Omron Sysmac Studio project Palletizing_Application_2 (Sysmac Studio 1.40.0.64008, StandardProject)

# Controller new_Controller_0: NJ501-1400 version 1.18
Units and slaves: Power Supply : NJ-Px3001; CPU : NJ501-1400
Task PrimaryTask (priority 4, period or condition 2000): TM_Modbus, TM_Movements_Connection, TM_Modbus_Connection, TM_Movements
Library TM_Commands 1.2.1 (contents left out)
Library TM_Modbus 1.1.0 (contents left out)

VAR_GLOBAL
    StartProgram : BOOL;
    CableConnected : BOOL;
    ListenNode_Connect_Connected : BOOL;
    ListenNode_Connect_TCP_Socket : _sSOCKET;
    MTCP_Connect_Connected : BOOL;
    MTCP_Connect_TCP_Socket : _sSOCKET;
END_VAR

PROGRAM TM_Modbus
VAR
    Enable : BOOL;
    DU_Enable : R_TRIG;
    NStep : INT;
    TON_Instance : TON;
    TM_Status_Instance : TM_Status;
    TM_Stop_Instance : TM_Stop;
    TM_ErrorCode_Instance : TM_ErrorCode;
    TM_PlayPause_Instance : TM_PlayPause;
    TM_ErrorCode_Execute : BOOL;
    TM_ErrorCode_Done : BOOL;
    TM_ErrorCode_Busy : BOOL;
    TM_ErrorCode_Error : BOOL;
    TM_ErrorCode_ErrorID : WORD;
    TM_Status_Execute : BOOL;
    TM_Status_Done : BOOL;
    TM_PlayPause_Execute : BOOL;
    TM_PlayPause_Done : BOOL;
    TM_PlayPause_Busy : BOOL;
    TM_PlayPause_Error : BOOL;
    TM_PlayPause_ErrorID : WORD;
    TM_Stop_Execute : BOOL;
    TM_Stop_Done : BOOL;
    TM_Stop_Busy : BOOL;
    TM_Stop_Error : BOOL;
    TM_Stop_ErrorID : WORD;
    TM_Status_Busy : BOOL;
    TM_Status_Error : BOOL;
    TM_Status_ErrorID : WORD;
    TM_ReadPosition_Instance : TM_ReadPosition;
    TM_ReadPosition_Execute : BOOL;
    TM_ReadPosition_Done : BOOL;
    TM_ReadPosition_Busy : BOOL;
    TM_ReadPosition_Error : BOOL;
    TM_ReadPosition_ErrorID : WORD;
    TM_ErrorCode_TMErrorCode : DINT;
    TM_Status_TMEditing : BOOL;
    TM_Status_TMError : BOOL;
    TM_Status_TMPaused : BOOL;
    TM_Status_TMRunning : BOOL;
    TM_PlayPauseButton : BOOL;
    TM_StopButton : BOOL;
    TM_ReadPosition_X : REAL;
    TM_ReadPosition_Y : REAL;
    TM_ReadPosition_Z : REAL;
    TM_ReadPosition_RX : REAL;
    TM_ReadPosition_RY : REAL;
    TM_ReadPosition_RZ : REAL;
END_VAR
VAR_EXTERNAL
    StartProgram : BOOL;
    CableConnected : BOOL;
    MTCP_Connect_TCP_Socket : _sSOCKET;
    MTCP_Connect_Connected : BOOL;
END_VAR
DU_Enable(Clk:=Enable);

Enable:=StartProgram;

IF DU_Enable.Q THEN
	
	NStep:=0;
	
END_IF;

IF Enable AND MTCP_Connect_Connected THEN
	
	CASE NStep OF
		
		0:
			IF TM_PlayPauseButton THEN
				NStep:=100;
			ELSIF TM_StopButton THEN
				NStep:=200;
			ELSE
				NStep:=300;
			END_IF;
		100:
			TM_PlayPause_Execute:=FALSE;
			TON_Instance.PT:=T#3s;
			TON_Instance.In:=FALSE;
			IF NOT TM_PlayPause_Done AND NOT TM_PlayPause_Error AND NOT TON_Instance.Q THEN
				NStep:=110;
			END_IF;
		110:
			TM_PlayPause_Execute:=TRUE;
			TON_Instance.In:=TRUE;
			IF TM_PlayPause_Done THEN
				CableConnected:=TRUE;
				TM_PlayPauseButton:=FALSE;
				NStep:=300;
			ELSIF (TM_PlayPause_Error AND (TM_PlayPause_ErrorID=16#2003 OR TM_PlayPause_ErrorID=16#2006)) THEN
				NStep:=300;
				CableConnected:=FALSE;
			ELSIF TON_Instance.Q THEN
				NStep:=100;
			END_IF;
		200:
			TM_Stop_Execute:=FALSE;
			TON_Instance.PT:=T#3s;
			TON_Instance.In:=FALSE;
			IF NOT TM_Stop_Done AND NOT TM_Stop_Error AND NOT TON_Instance.Q THEN
				NStep:=210;
			END_IF;
		210:
			TM_Stop_Execute:=TRUE;
			TON_Instance.In:=TRUE;
			IF TM_Stop_Done THEN
				TM_StopButton:=FALSE;
				CableConnected:=TRUE;
				NStep:=300;
			ELSIF (TM_Stop_Error AND (TM_Stop_ErrorID=16#2003 OR TM_Stop_ErrorID=16#2006)) THEN
				NStep:=300;
				CableConnected:=FALSE;
			ELSIF TON_Instance.Q THEN
				NStep:=200;
			END_IF;
		300:
			TM_Status_Execute:=FALSE;
			TON_Instance.PT:=T#3s;
			TON_Instance.In:=FALSE;
			IF NOT TM_Status_Done AND NOT TM_Status_Error AND NOT TON_Instance.Q THEN
				NStep:=310;
			END_IF;
		310:
			TM_Status_Execute:=TRUE;
			TON_Instance.In:=TRUE;
			IF TM_Status_Done THEN
				NStep:=400;
				CableConnected:=TRUE;
			ELSIF TM_Status_Error AND (TM_Status_ErrorID=16#2003 OR  TM_Status_ErrorID=16#2006) THEN
				NStep:=300;
				CableConnected:=FALSE;
			ELSIF TON_Instance.Q THEN
				NStep:=300;
			END_IF;
		400:
			TM_ErrorCode_Execute:=FALSE;
			TON_Instance.PT:=T#3s;
			TON_Instance.In:=FALSE;
			IF NOT TM_ErrorCode_Done AND NOT TM_ErrorCode_Error AND NOT TON_Instance.Q THEN
				NStep:=410;
			END_IF;
		410:
			TM_ErrorCode_Execute:=TRUE;
			TON_Instance.In:=TRUE;
			IF TM_ErrorCode_Done THEN
				CableConnected:=TRUE;
				NStep:=500;
			ELSIF (TM_ErrorCode_Error AND (TM_ErrorCode_ErrorID=16#2003 OR TM_ErrorCode_ErrorID=16#2006)) THEN
				NStep:=400;
				CableConnected:=FALSE;
			ELSIF TON_Instance.Q THEN
				NStep:=400;
			END_IF;
		500:
			TM_ReadPosition_Execute:=FALSE;
			TON_Instance.PT:=T#3s;
			TON_Instance.In:=FALSE;
			IF NOT TM_ReadPosition_Done AND NOT TM_ReadPosition_Error AND NOT TON_Instance.Q THEN
				NStep:=510;
			END_IF;
		510:
			TM_ReadPosition_Execute:=TRUE;
			TON_Instance.In:=TRUE;
			IF TM_ReadPosition_Done THEN
				CableConnected:=TRUE;
				NStep:=600;
			ELSIF (TM_ReadPosition_Error AND (TM_ReadPosition_ErrorID=16#2003 OR TM_ReadPosition_ErrorID=16#2006)) THEN
				NStep:=500;
				CableConnected:=FALSE;
			ELSIF TON_Instance.Q THEN
				NStep:=500;
			END_IF;
		600:
			TON_Instance.In:=FALSE;
			TON_Instance.PT:=T#1s;
			IF (NOT TON_Instance.Q) THEN
				NStep:=610;
			END_IF;
		610:
			TON_Instance.In:=TRUE;
			IF TON_Instance.Q THEN
				NStep:=0;
			END_IF;		
		
	END_CASE;
	
END_IF;

TON_Instance();

TM_ErrorCode_Instance(
	Execute:=TM_ErrorCode_Execute,
	Socket:=MTCP_Connect_TCP_Socket,
	Done=>TM_ErrorCode_Done,
	TMErrorCode=>TM_ErrorCode_TMErrorCode,
	Busy=>TM_ErrorCode_Busy,
	Error=>TM_ErrorCode_Error,
	ErrorID=>TM_ErrorCode_ErrorID
);

TM_Status_Instance(
	Execute:=TM_Status_Execute,
	Socket:=MTCP_Connect_TCP_Socket,
	Done=>TM_Status_Done,
	TMRunning=>TM_Status_TMRunning,
	TMEditing=>TM_Status_TMEditing,
	TMError=>TM_Status_TMError,
	TMPaused=>TM_Status_TMPaused,
	Busy=>TM_Status_Busy,
	Error=>TM_Status_Error,
	ErrorID=>TM_Status_ErrorID
);

TM_PlayPause_Instance(
	Execute:=TM_PlayPause_Execute,
	Socket:=MTCP_Connect_TCP_Socket,
	Done=>TM_PlayPause_Done,
	Busy=>TM_PlayPause_Busy,
	Error=>TM_PlayPause_Error,
	ErrorID=>TM_PlayPause_ErrorID
);

TM_Stop_Instance(
	Execute:=TM_Stop_Execute,
	Socket:=MTCP_Connect_TCP_Socket,
	Done=>TM_Stop_Done,
	Busy=>TM_Stop_Busy,
	Error=>TM_Stop_Error,
	ErrorID=>TM_Stop_ErrorID
);

TM_ReadPosition_Instance(
	Execute:=TM_ReadPosition_Execute,
	Socket:=MTCP_Connect_TCP_Socket,
	Done=>TM_ReadPosition_Done,
	Busy=>TM_ReadPosition_Busy,
	Error=>TM_ReadPosition_Error,
	ErrorID=>TM_ReadPosition_ErrorID,
	X=>TM_ReadPosition_X,
	Y=>TM_ReadPosition_Y,
	Z=>TM_ReadPosition_Z,
	RX=>TM_ReadPosition_RX,
	RY=>TM_ReadPosition_RY,
	RZ=>TM_ReadPosition_RZ
);
END_PROGRAM

PROGRAM TM_Movements_Connection
VAR
    ListenNode_Connect_Instance : ListenNode_Connect;
    ListenNode_Connect_Enable : BOOL;
    ListenNode_Connect_IPaddress : STRING[16];
    ListenNode_Connect_Port : UINT;
    ListenNode_Connect_Connect : BOOL;
    ListenNode_Connect_Error : BOOL;
    ListenNode_Connect_ErrorID : WORD;
    ListenNode_Connect_EtnConnError : BOOL;
    ListenNode_Connect_Socket_Status : _eCONNECTION_STATE;
END_VAR
VAR_EXTERNAL
    ListenNode_Connect_Connected : BOOL;
    ListenNode_Connect_TCP_Socket : _sSOCKET;
    StartProgram : BOOL;
END_VAR
ListenNode_Connect_Enable:=TRUE;
ListenNode_Connect_IPaddress:='192.168.250.30';
ListenNode_Connect_Port:=5890;

ListenNode_Connect_Connect:=StartProgram;

ListenNode_Connect_Instance(
	Enable:=ListenNode_Connect_Enable,
	IPaddress:=ListenNode_Connect_IPaddress,
	Port:=ListenNode_Connect_Port,
	Connect:=ListenNode_Connect_Connect,
	Connected=>ListenNode_Connect_Connected,
	Error=>ListenNode_Connect_Error,
	ErrorID=>ListenNode_Connect_ErrorID,
	EtnConnError=>ListenNode_Connect_EtnConnError,
	TCP_Socket=>ListenNode_Connect_TCP_Socket,
	Socket_Status=>ListenNode_Connect_Socket_Status
);
END_PROGRAM

PROGRAM TM_Modbus_Connection
VAR
    MTCP_Connect_Instance : MTCP_Connect;
    MTCP_Connect_Enable : BOOL;
    MTCP_Connect_Port : UINT;
    MTCP_Connect_Connect : BOOL;
    MTCP_Connect_Error : BOOL;
    MTCP_Connect_ErrorID : WORD;
    MTCP_Connect_EtnConnError : BOOL;
    MTCP_Connect_Socket_Status : _eCONNECTION_STATE;
    MTCP_Connect_IPaddress : STRING[16];
END_VAR
VAR_EXTERNAL
    StartProgram : BOOL;
    MTCP_Connect_Connected : BOOL;
    MTCP_Connect_TCP_Socket : _sSOCKET;
END_VAR
MTCP_Connect_Enable:=TRUE;
MTCP_Connect_IPaddress:='192.168.250.30';
MTCP_Connect_Port:=502;

MTCP_Connect_Connect:=StartProgram;

MTCP_Connect_Instance(
	Enable:=MTCP_Connect_Enable,
	IPaddress:=MTCP_Connect_IPaddress,
	Port:=MTCP_Connect_Port,
	Connect:=MTCP_Connect_Connect,
	Connected=>MTCP_Connect_Connected,
	Error=>MTCP_Connect_Error,
	ErrorID=>MTCP_Connect_ErrorID,
	EtnConnError=>MTCP_Connect_EtnConnError,
	TCP_Socket=>MTCP_Connect_TCP_Socket,
	Socket_Status=>MTCP_Connect_Socket_Status
);
END_PROGRAM

PROGRAM TM_Movements
VAR
    TM_ChangeLoad_Instance : TM_ChangeLoad;
    TM_ChangeTCP_Instance : TM_ChangeTCP;
    TM_MovCmd_Instance : TM_MovCmd;
    TM_MovCmd_Done : BOOL;
    TM_MovCmd_Busy : BOOL;
    TM_MovCmd_Error : BOOL;
    TM_MovCmd_ErrorID : WORD;
    TM_MovCmd_Execute : BOOL;
    TM_MovCmd_Movement : STRING[256];
    TM_MovCmd_DataFormat : STRING[256];
    DD_ListenNode_Connect_Connected : F_TRIG;
    TM_MovCmd_Point : STRING[256];
    TM_MovCmd_Speed : INT;
    TM_MovCmd_AccelTime : INT;
    TM_MovCmd_Blending : INT;
    TM_MovCmd_PrecisePos : BOOL;
    TM_MovCmd_RobotPose : STRING[256];
    TM_MovCmd_Command : STRING[256];
    TM_MovCmd_ActivateExit : BOOL;
    TM_MovCmd_CommandID : INT;
    Enable : BOOL;
    DU_Enable : R_TRIG;
    TM_ChangeBase_Busy : BOOL;
    TM_ChangeBase_Done : BOOL;
    TM_ChangeBase_Error : BOOL;
    TM_ChangeBase_ErrorID : WORD;
    TM_ChangeBase_Execute : BOOL;
    TM_ChangeBase_Base : STRING[256];
    TM_ChangeBase_ActivateExit : BOOL;
    TM_ChangeBase_CommandID : INT;
    TM_ChangeLoad_Execute : BOOL;
    TM_ChangeLoad_Busy : BOOL;
    TM_ChangeLoad_Done : BOOL;
    TM_ChangeLoad_Error : BOOL;
    TM_ChangeLoad_ErrorID : WORD;
    TM_ChangeLoad_Payload : STRING[256];
    TM_ChangeLoad_ActivateExit : BOOL;
    TM_ChangeLoad_CommandID : INT;
    TM_ChangeTCP_Busy : BOOL;
    TM_ChangeTCP_Done : BOOL;
    TM_ChangeTCP_Error : BOOL;
    TM_ChangeTCP_ErrorID : WORD;
    TM_ChangeTCP_Execute : BOOL;
    TM_ChangeTCP_TCP : STRING[256];
    TM_ChangeTCP_Weight : STRING[256];
    TM_ChangeTCP_MomInertia : STRING[256];
    TM_ChangeTCP_RefFrame : STRING[256];
    TM_ChangeTCP_ActivateExit : BOOL;
    TM_ChangeTCP_CommandID : INT;
    TM_CircleCmd_Done : BOOL;
    TM_CircleCmd_Busy : BOOL;
    TM_CircleCmd_Error : BOOL;
    TM_CircleCmd_ErrorID : WORD;
    TM_CircleCmd_Execute : BOOL;
    TM_CircleCmd_DataFormat : STRING[256];
    TM_CircleCmd_ArcPoint : STRING[256];
    TM_CircleCmd_EndArcPoint : STRING[256];
    TM_CircleCmd_Speed : INT;
    TM_CircleCmd_AccelTime : INT;
    TM_CircleCmd_Blending : INT;
    TM_CircleCmd_ArcAngle : INT;
    TM_CircleCmd_PrecisePos : BOOL;
    TM_CircleCmd_Command : STRING[256];
    TM_CircleCmd_ActivateExit : BOOL;
    TM_CircleCmd_CommandID : INT;
    PickPoint : STRING[256];
    PalletFirstPoint : STRING[256];
    StartPoint : STRING[256];
    PalletSecondPoint : STRING[256];
    PalletThirdPoint : STRING[256];
    PalletFourthPoint : STRING[256];
    MovementIndicatorStage : INT;
    DownRelative : STRING[256];
    HighRelative : STRING[256];
    TM_ChangeBase_Command : STRING[256];
    TM_ChangeLoad_Command : STRING[256];
    TM_ChangeTCP_Command : STRING[256];
    DD_CableConnected : F_TRIG;
    TM_MovCmd_ListenNode : STRING[256];
    Stage : INT;
    TM_MovCmd_TimeOutET : TIME;
    TM_MovCmd_Enable : BOOL;
    TM_ChangeTCP_Enable : BOOL;
    TM_ChangeTCP_ListenNode : STRING[256];
    TM_ChangeTCP_TimeOutET : TIME;
    TM_ChangeLoad_Enable : BOOL;
    TM_ChangeLoad_ListenNode : STRING[256];
    TM_ChangeLoad_TimeOutET : TIME;
    TM_CircleCmd_Instance : TM_CircleCmd;
    TM_ChangeBase_Instance : TM_ChangeBase;
    TM_ChangeBase_Enable : BOOL;
    TM_CircleCmd_Enable : BOOL;
    TM_CircleCmd_ListenNode : STRING[256];
    TM_CircleCmd_TimeOutET : TIME;
    TM_ChangeBase_ListenNode : STRING[256];
    TM_ChangeBase_TimeOutET : TIME;
END_VAR
VAR_EXTERNAL
    StartProgram : BOOL;
    CableConnected : BOOL;
    ListenNode_Connect_Connected : BOOL;
    ListenNode_Connect_TCP_Socket : _sSOCKET;
END_VAR
DU_Enable(Clk:=Enable);
DD_ListenNode_Connect_Connected(Clk:=ListenNode_Connect_Connected);
DD_CableConnected(Clk:=CableConnected);

Enable:=StartProgram;

IF DU_Enable.Q THEN
	
	Stage:=0;
	MovementIndicatorStage:=0;
	
	PickPoint:='400,100,400,180,0,90';
	PalletFirstPoint:='200,-200,400,180,0,90';
	PalletSecondPoint:='200,-400,400,180,0,90';
	PalletThirdPoint:='400,-200,400,180,0,90';
	PalletFourthPoint:='400,-400,400,180,0,90';
	StartPoint:='400,0,500,150,0,90';
	DownRelative:='0,0,-100,0,0,0';
	HighRelative:='0,0,100,0,0,0';
	
END_IF;

IF DD_ListenNode_Connect_Connected.Q OR DD_CableConnected.Q THEN //connection closed or cable disconnected.
	
	Stage:=MovementIndicatorStage;
	
END_IF;

IF Enable AND ListenNode_Connect_Connected AND CableConnected THEN	//the PLC program is enabled and there is connection with listen node and the cable is connected
	
	CASE Stage OF
		
		//-----------------------------------------------------------TCP Selection--------------------------------------------------
		0:
			TM_ChangeTCP_Enable:=FALSE;
			IF (NOT TM_ChangeTCP_Done) AND (NOT TM_ChangeTCP_Error) AND (NOT TM_ChangeTCP_Busy) THEN
				Stage:=1; 
			END_IF;
		1:
			TM_ChangeTCP_Enable:=TRUE;	
			TM_ChangeTCP_ActivateExit:=TRUE;
			TM_ChangeTCP_CommandID:=1;
			TM_ChangeTCP_Execute:=FALSE;
			TM_ChangeTCP_ListenNode:='Listen1';
			TM_ChangeTCP_TCP:='DefinedTool';
			TM_ChangeTCP_Command:='var_i=10';
			TM_ChangeTCP_Weight:='';
			TM_ChangeTCP_MomInertia:='';
			TM_ChangeTCP_RefFrame:='';
			TM_ChangeLoad_Payload:='';
			IF (NOT TM_ChangeTCP_Done) AND (NOT TM_ChangeTCP_Error) THEN
				Stage:=2;
			END_IF;
		2:
			TM_ChangeTCP_Execute:=TRUE;
			IF TM_ChangeTCP_Done THEN
				Stage:=10;
			ELSIF TM_ChangeTCP_Error THEN
				Stage:=9999;
			END_IF;
		//-----------------------------------------------------------Program Stages--------------------------------------------------------------
		10:
			TM_MovCmd_Enable:=FALSE;
			MovementIndicatorStage:=Stage;
			IF (NOT TM_MovCmd_Done) AND (NOT TM_MovCmd_Error) AND (NOT TM_MovCmd_Busy) THEN
				Stage:=11;
			END_IF;
		11:
			TM_MovCmd_Enable:=TRUE;
			TM_MovCmd_Movement:='PTP';
			TM_MovCmd_DataFormat:='CPP';
			TM_MovCmd_Point:=StartPoint;
			TM_MovCmd_Speed:=30;
			TM_MovCmd_AccelTime:=200;
			TM_MovCmd_Blending:=100;
			TM_MovCmd_PrecisePos:=1;
			TM_MovCmd_RobotPose:='';
			TM_MovCmd_Command:='var_i=40';
			TM_MovCmd_ActivateExit:=TRUE;
			TM_MovCmd_CommandID:=1;
			TM_MovCmd_Execute:=FALSE;
			TM_MovCmd_ListenNode:='Listen1';
			IF (NOT TM_MovCmd_Done) AND (NOT TM_MovCmd_Error) THEN
				Stage:=12;
			END_IF;
		12:
			TM_MovCmd_Execute:=TRUE;
			IF TM_MovCmd_Done THEN
				Stage:=20;
			ELSIF TM_MovCmd_Error THEN
				Stage:=9999;
			END_IF;
		20:
			TM_MovCmd_Enable:=FALSE;
			MovementIndicatorStage:=Stage;
			IF (NOT TM_MovCmd_Done) AND (NOT TM_MovCmd_Error) AND (NOT TM_MovCmd_Busy) THEN
				Stage:=21;
			END_IF;
		21:			
			TM_MovCmd_Enable:=TRUE;
			TM_MovCmd_Movement:='Line';
			TM_MovCmd_DataFormat:='CPR';
			TM_MovCmd_Point:=StartPoint;
			TM_MovCmd_Speed:=30;
			TM_MovCmd_AccelTime:=200;
			TM_MovCmd_Blending:=100;
			TM_MovCmd_PrecisePos:=1;
			TM_MovCmd_RobotPose:='';
			TM_MovCmd_Command:='var_i=30';
			TM_MovCmd_ActivateExit:=TRUE;
			TM_MovCmd_CommandID:=1;
			TM_MovCmd_Execute:=FALSE;
			TM_MovCmd_ListenNode:='Listen1';
			IF (NOT TM_MovCmd_Done) AND (NOT TM_MovCmd_Error) THEN
				Stage:=22;
			END_IF;	
		22:
			TM_MovCmd_Execute:=TRUE;
			IF TM_MovCmd_Done THEN
				Stage:=30;
			ELSIF TM_MovCmd_Error THEN
				Stage:=9999;
			END_IF;
		30:
			TM_MovCmd_Enable:=FALSE;
			MovementIndicatorStage:=Stage;
			IF (NOT TM_MovCmd_Done) AND (NOT TM_MovCmd_Error) AND (NOT TM_MovCmd_Busy) THEN
				Stage:=31;
			END_IF;
		31:			
			TM_MovCmd_Enable:=TRUE;
			TM_MovCmd_Movement:='Line';
			TM_MovCmd_DataFormat:='CPR';
			TM_MovCmd_Point:=PickPoint;
			TM_MovCmd_Speed:=30;
			TM_MovCmd_AccelTime:=200;
			TM_MovCmd_Blending:=100;
			TM_MovCmd_PrecisePos:=1;
			TM_MovCmd_RobotPose:='';
			TM_MovCmd_Command:='var_i=10';
			TM_MovCmd_ActivateExit:=FALSE;
			TM_MovCmd_CommandID:=1;
			TM_MovCmd_Execute:=FALSE;
			TM_MovCmd_ListenNode:='Listen1';
			IF (NOT TM_MovCmd_Done) AND (NOT TM_MovCmd_Error) THEN
				Stage:=32;
			END_IF;			
		32:
			TM_MovCmd_Execute:=TRUE;
			IF TM_MovCmd_Done THEN
				Stage:=40;
			ELSIF TM_MovCmd_Error THEN
				Stage:=9999;
			END_IF;
		40:
			TM_MovCmd_Enable:=FALSE;
			IF (NOT TM_MovCmd_Done) AND (NOT TM_MovCmd_Error) AND (NOT TM_MovCmd_Busy) THEN
				Stage:=41;
			END_IF;
		41:			
			TM_MovCmd_Enable:=TRUE;
			TM_MovCmd_Movement:='Move_Line';
			TM_MovCmd_DataFormat:='CPP';
			TM_MovCmd_Point:=DownRelative;
			TM_MovCmd_Speed:=30;
			TM_MovCmd_AccelTime:=200;
			TM_MovCmd_Blending:=100;
			TM_MovCmd_PrecisePos:=1;
			TM_MovCmd_RobotPose:='';
			TM_MovCmd_Command:='var_i=10';
			TM_MovCmd_ActivateExit:=TRUE;
			TM_MovCmd_CommandID:=2;
			TM_MovCmd_Execute:=FALSE;
			TM_MovCmd_ListenNode:='Listen1';
			IF (NOT TM_MovCmd_Done) AND (NOT TM_MovCmd_Error) THEN
				Stage:=42;
			END_IF;
		42:
			TM_MovCmd_Execute:=TRUE;
			IF TM_MovCmd_Done THEN
				Stage:=50;
			ELSIF TM_MovCmd_Error THEN
				Stage:=9999;
			END_IF;
		50:
			TM_ChangeLoad_Enable:=FALSE;
			IF (NOT TM_ChangeLoad_Done) AND (NOT TM_ChangeLoad_Error) AND (NOT TM_ChangeLoad_Busy) THEN
				Stage:=51;
			END_IF;
		51:
			TM_ChangeLoad_Enable:=TRUE;	 
			TM_ChangeLoad_ActivateExit:=TRUE;
			TM_ChangeLoad_CommandID:=1;
			TM_ChangeLoad_Execute:=FALSE;
			TM_ChangeLoad_ListenNode:='Listen1';
			TM_ChangeLoad_Command:='var_i=20';
			TM_ChangeLoad_Payload:='0.2';
			IF (NOT TM_ChangeLoad_Done) AND (NOT TM_ChangeLoad_Error) THEN
				Stage:=52;
			END_IF;
		52:
			TM_ChangeLoad_Execute:=TRUE;
			IF TM_ChangeLoad_Done THEN
				Stage:=60;
			ELSIF TM_ChangeLoad_Error THEN
				Stage:=9999;
			END_IF;			
		60:
			TM_MovCmd_Enable:=FALSE;
			IF (NOT TM_MovCmd_Done) AND (NOT TM_MovCmd_Error) AND (NOT TM_MovCmd_Busy) THEN
				Stage:=61;
			END_IF;	
		61:
			TM_MovCmd_Enable:=TRUE;
			TM_MovCmd_Movement:='Move_Line';
			TM_MovCmd_DataFormat:='CPP';
			TM_MovCmd_Point:=HighRelative;
			TM_MovCmd_Speed:=30;
			TM_MovCmd_AccelTime:=200;
			TM_MovCmd_Blending:=100;
			TM_MovCmd_PrecisePos:=1;
			TM_MovCmd_RobotPose:='';
			TM_MovCmd_Command:='var_i=10';
			TM_MovCmd_ActivateExit:=TRUE;
			TM_MovCmd_CommandID:=2;
			TM_MovCmd_Execute:=FALSE;
			TM_MovCmd_ListenNode:='Listen1';
			IF (NOT TM_MovCmd_Done) AND (NOT TM_MovCmd_Error) THEN
				Stage:=62;
			END_IF;
		62:
			TM_MovCmd_Execute:=TRUE;
			IF TM_MovCmd_Done THEN
				Stage:=70;
			ELSIF TM_MovCmd_Error THEN
				Stage:=9999;
			END_IF;
		70:
			TM_MovCmd_Enable:=FALSE;
			MovementIndicatorStage:=Stage;
			IF (NOT TM_MovCmd_Done) AND (NOT TM_MovCmd_Error) AND (NOT TM_MovCmd_Busy) THEN
				Stage:=71;
			END_IF;	
		71:
			TM_MovCmd_Enable:=TRUE;
			TM_MovCmd_Movement:='Line';
			TM_MovCmd_DataFormat:='CPR';
			TM_MovCmd_Point:=PalletFirstPoint;
			TM_MovCmd_Speed:=30;
			TM_MovCmd_AccelTime:=200;
			TM_MovCmd_Blending:=100;
			TM_MovCmd_PrecisePos:=1;
			TM_MovCmd_RobotPose:='';
			TM_MovCmd_Command:='var_i=10';
			TM_MovCmd_ActivateExit:=FALSE;
			TM_MovCmd_CommandID:=1;
			TM_MovCmd_Execute:=FALSE;
			TM_MovCmd_ListenNode:='Listen1';
			IF (NOT TM_MovCmd_Done) AND (NOT TM_MovCmd_Error) THEN
				Stage:=72;
			END_IF;
		72:
			TM_MovCmd_Execute:=TRUE;
			IF TM_MovCmd_Done THEN
				Stage:=80;
			ELSIF TM_MovCmd_Error THEN
				Stage:=9999;
			END_IF;
		80:
			TM_MovCmd_Enable:=FALSE;
			IF (NOT TM_MovCmd_Done) AND (NOT TM_MovCmd_Error) AND (NOT TM_MovCmd_Busy) THEN
				Stage:=81;
			END_IF;	
		81:
			TM_MovCmd_Enable:=TRUE;
			TM_MovCmd_Movement:='Move_Line';
			TM_MovCmd_DataFormat:='CPP';
			TM_MovCmd_Point:=DownRelative;
			TM_MovCmd_Speed:=30;
			TM_MovCmd_AccelTime:=200;
			TM_MovCmd_Blending:=100;
			TM_MovCmd_PrecisePos:=1;
			TM_MovCmd_RobotPose:='';
			TM_MovCmd_Command:='var_i=10';
			TM_MovCmd_ActivateExit:=TRUE;
			TM_MovCmd_CommandID:=2;
			TM_MovCmd_Execute:=FALSE;
			TM_MovCmd_ListenNode:='Listen1';
			IF (NOT TM_MovCmd_Done) AND (NOT TM_MovCmd_Error) THEN
				Stage:=82;
			END_IF;
		82:
			TM_MovCmd_Execute:=TRUE;
			IF TM_MovCmd_Done THEN
				Stage:=90;
			ELSIF TM_MovCmd_Error THEN
				Stage:=9999;
			END_IF;
		90:
			TM_ChangeLoad_Enable:=FALSE;
			IF (NOT TM_ChangeLoad_Done) AND (NOT TM_ChangeLoad_Error) AND (NOT TM_ChangeLoad_Busy) THEN
				Stage:=91;
			END_IF;
		91:
			TM_ChangeLoad_Enable:=TRUE;	 
			TM_ChangeLoad_ActivateExit:=TRUE;
			TM_ChangeLoad_CommandID:=1;
			TM_ChangeLoad_Execute:=FALSE;
			TM_ChangeLoad_ListenNode:='Listen1';
			TM_ChangeLoad_Command:='var_i=30';
			TM_ChangeLoad_Payload:='0';
			IF (NOT TM_ChangeLoad_Done) AND (NOT TM_ChangeLoad_Error) THEN
				Stage:=92;
			END_IF;
		92:
			TM_ChangeLoad_Execute:=TRUE;
			IF TM_ChangeLoad_Done THEN
				Stage:=100;
			ELSIF TM_ChangeLoad_Error THEN
				Stage:=9999;
			END_IF;
		100:
			TM_MovCmd_Enable:=FALSE;
			IF (NOT TM_MovCmd_Done) AND (NOT TM_MovCmd_Error) AND (NOT TM_MovCmd_Busy) THEN
				Stage:=101;
			END_IF;	
		101:
			TM_MovCmd_Enable:=TRUE;
			TM_MovCmd_Movement:='Move_Line';
			TM_MovCmd_DataFormat:='CPP';
			TM_MovCmd_Point:=HighRelative;
			TM_MovCmd_Speed:=30;
			TM_MovCmd_AccelTime:=200;
			TM_MovCmd_Blending:=100;
			TM_MovCmd_PrecisePos:=1;
			TM_MovCmd_RobotPose:='';
			TM_MovCmd_Command:='var_i=10';
			TM_MovCmd_ActivateExit:=TRUE;
			TM_MovCmd_CommandID:=2;
			TM_MovCmd_Execute:=FALSE;
			TM_MovCmd_ListenNode:='Listen1';
			IF (NOT TM_MovCmd_Done) AND (NOT TM_MovCmd_Error) THEN
				Stage:=102;
			END_IF;
		102:
			TM_MovCmd_Execute:=TRUE;
			IF TM_MovCmd_Done THEN
				Stage:=110;
			ELSIF TM_MovCmd_Error THEN
				Stage:=9999;
			END_IF;
		110:
			TM_MovCmd_Enable:=FALSE;
			MovementIndicatorStage:=Stage;
			IF (NOT TM_MovCmd_Done) AND (NOT TM_MovCmd_Error) AND (NOT TM_MovCmd_Busy) THEN
				Stage:=111;
			END_IF;	
		111:
			TM_MovCmd_Enable:=TRUE;
			TM_MovCmd_Movement:='Line';
			TM_MovCmd_DataFormat:='CPR';
			TM_MovCmd_Point:=PickPoint;
			TM_MovCmd_Speed:=30;
			TM_MovCmd_AccelTime:=200;
			TM_MovCmd_Blending:=100;
			TM_MovCmd_PrecisePos:=1;
			TM_MovCmd_RobotPose:='';
			TM_MovCmd_Command:='var_i=10';
			TM_MovCmd_ActivateExit:=FALSE;
			TM_MovCmd_CommandID:=1;
			TM_MovCmd_Execute:=FALSE;
			TM_MovCmd_ListenNode:='Listen1';
			IF (NOT TM_MovCmd_Done) AND (NOT TM_MovCmd_Error) THEN
				Stage:=112;
			END_IF;
		112:
			TM_MovCmd_Execute:=TRUE;
			IF TM_MovCmd_Done THEN
				Stage:=120;
			ELSIF TM_MovCmd_Error THEN
				Stage:=9999;
			END_IF;
		120:
			TM_MovCmd_Enable:=FALSE;
			IF (NOT TM_MovCmd_Done) AND (NOT TM_MovCmd_Error) AND (NOT TM_MovCmd_Busy) THEN
				Stage:=121;
			END_IF;	
		121:
			TM_MovCmd_Enable:=TRUE;
			TM_MovCmd_Movement:='Move_Line';
			TM_MovCmd_DataFormat:='CPP';
			TM_MovCmd_Point:=DownRelative;
			TM_MovCmd_Speed:=30;
			TM_MovCmd_AccelTime:=200;
			TM_MovCmd_Blending:=100;
			TM_MovCmd_PrecisePos:=1;
			TM_MovCmd_RobotPose:='';
			TM_MovCmd_Command:='var_i=10';
			TM_MovCmd_ActivateExit:=TRUE;
			TM_MovCmd_CommandID:=2;
			TM_MovCmd_Execute:=FALSE;
			TM_MovCmd_ListenNode:='Listen1';
			IF (NOT TM_MovCmd_Done) AND (NOT TM_MovCmd_Error) THEN
				Stage:=122;
			END_IF;
		122:
			TM_MovCmd_Execute:=TRUE;
			IF TM_MovCmd_Done THEN
				Stage:=130;
			ELSIF TM_MovCmd_Error THEN
				Stage:=9999;
			END_IF;
		130:
			TM_ChangeLoad_Enable:=FALSE;
			IF (NOT TM_ChangeLoad_Done) AND (NOT TM_ChangeLoad_Error) AND (NOT TM_ChangeLoad_Busy) THEN
				Stage:=131;
			END_IF;
		131:
			TM_ChangeLoad_Enable:=TRUE;	 
			TM_ChangeLoad_ActivateExit:=TRUE;
			TM_ChangeLoad_CommandID:=1;
			TM_ChangeLoad_Execute:=FALSE;
			TM_ChangeLoad_ListenNode:='Listen1';
			TM_ChangeLoad_Command:='var_i=20';
			TM_ChangeLoad_Payload:='0.2';
			IF (NOT TM_ChangeLoad_Done) AND (NOT TM_ChangeLoad_Error) THEN
				Stage:=132;
			END_IF;
		132:
			TM_ChangeLoad_Execute:=TRUE;
			IF TM_ChangeLoad_Done THEN
				Stage:=140;
			ELSIF TM_ChangeLoad_Error THEN
				Stage:=9999;
			END_IF;
		140:
			TM_MovCmd_Enable:=FALSE;
			IF (NOT TM_MovCmd_Done) AND (NOT TM_MovCmd_Error) AND (NOT TM_MovCmd_Busy) THEN
				Stage:=141;
			END_IF;
		141:
			TM_MovCmd_Enable:=TRUE;
			TM_MovCmd_Movement:='Move_Line';
			TM_MovCmd_DataFormat:='CPP';
			TM_MovCmd_Point:=HighRelative;
			TM_MovCmd_Speed:=30;
			TM_MovCmd_AccelTime:=200;
			TM_MovCmd_Blending:=100;
			TM_MovCmd_PrecisePos:=1;
			TM_MovCmd_RobotPose:='';
			TM_MovCmd_Command:='var_i=10';
			TM_MovCmd_ActivateExit:=TRUE;
			TM_MovCmd_CommandID:=2;
			TM_MovCmd_Execute:=FALSE;
			TM_MovCmd_ListenNode:='Listen1';
			IF (NOT TM_MovCmd_Done) AND (NOT TM_MovCmd_Error) THEN
				Stage:=142;
			END_IF;
		142:
			TM_MovCmd_Execute:=TRUE;
			IF TM_MovCmd_Done THEN
				Stage:=150;
			ELSIF TM_MovCmd_Error THEN
				Stage:=9999;
			END_IF;
		150:
			TM_MovCmd_Enable:=FALSE;
			MovementIndicatorStage:=Stage;
			IF (NOT TM_MovCmd_Done) AND (NOT TM_MovCmd_Error) AND (NOT TM_MovCmd_Busy) THEN
				Stage:=151;
			END_IF;
		151:
			TM_MovCmd_Enable:=TRUE;
			TM_MovCmd_Movement:='Line';
			TM_MovCmd_DataFormat:='CPR';
			TM_MovCmd_Point:=PalletSecondPoint;
			TM_MovCmd_Speed:=30;
			TM_MovCmd_AccelTime:=200;
			TM_MovCmd_Blending:=100;
			TM_MovCmd_PrecisePos:=1;
			TM_MovCmd_RobotPose:='';
			TM_MovCmd_Command:='var_i=10';
			TM_MovCmd_ActivateExit:=FALSE;
			TM_MovCmd_CommandID:=1;
			TM_MovCmd_Execute:=FALSE;
			TM_MovCmd_ListenNode:='Listen1';
			IF (NOT TM_MovCmd_Done) AND (NOT TM_MovCmd_Error) THEN
				Stage:=152;
			END_IF;
		152:
			TM_MovCmd_Execute:=TRUE;
			IF TM_MovCmd_Done THEN
				Stage:=160;
			ELSIF TM_MovCmd_Error THEN
				Stage:=9999;
			END_IF;
		160:
			TM_MovCmd_Enable:=FALSE;
			IF (NOT TM_MovCmd_Done) AND (NOT TM_MovCmd_Error) AND (NOT TM_MovCmd_Busy) THEN
				Stage:=161;
			END_IF;	
		161:
			TM_MovCmd_Enable:=TRUE;
			TM_MovCmd_Movement:='Move_Line';
			TM_MovCmd_DataFormat:='CPP';
			TM_MovCmd_Point:=DownRelative;
			TM_MovCmd_Speed:=30;
			TM_MovCmd_AccelTime:=200;
			TM_MovCmd_Blending:=100;
			TM_MovCmd_PrecisePos:=1;
			TM_MovCmd_RobotPose:='';
			TM_MovCmd_Command:='var_i=10';
			TM_MovCmd_ActivateExit:=TRUE;
			TM_MovCmd_CommandID:=2;
			TM_MovCmd_Execute:=FALSE;
			TM_MovCmd_ListenNode:='Listen1';
			IF (NOT TM_MovCmd_Done) AND (NOT TM_MovCmd_Error) THEN
				Stage:=162;
			END_IF;
		162:
			TM_MovCmd_Execute:=TRUE;
			IF TM_MovCmd_Done THEN
				Stage:=170;
			ELSIF TM_MovCmd_Error THEN
				Stage:=9999;
			END_IF;
		170:
			TM_ChangeLoad_Enable:=FALSE;
			IF (NOT TM_ChangeLoad_Done) AND (NOT TM_ChangeLoad_Error) AND (NOT TM_ChangeLoad_Busy) THEN
				Stage:=171;
			END_IF;
		171:
			TM_ChangeLoad_Enable:=TRUE;	 
			TM_ChangeLoad_ActivateExit:=TRUE;
			TM_ChangeLoad_CommandID:=1;
			TM_ChangeLoad_Execute:=FALSE;
			TM_ChangeLoad_ListenNode:='Listen1';
			TM_ChangeLoad_Command:='var_i=30';
			TM_ChangeLoad_Payload:='0';
			IF (NOT TM_ChangeLoad_Done) AND (NOT TM_ChangeLoad_Error) THEN
				Stage:=172;
			END_IF;
		172:
			TM_ChangeLoad_Execute:=TRUE;
			IF TM_ChangeLoad_Done THEN
				Stage:=180;
			ELSIF TM_ChangeLoad_Error THEN
				Stage:=9999;
			END_IF;
		180:
			TM_MovCmd_Enable:=FALSE;
			IF (NOT TM_MovCmd_Done) AND (NOT TM_MovCmd_Error) AND (NOT TM_MovCmd_Busy) THEN
				Stage:=181;
			END_IF;	
		181:
			TM_MovCmd_Enable:=TRUE;
			TM_MovCmd_Movement:='Move_Line';
			TM_MovCmd_DataFormat:='CPP';
			TM_MovCmd_Point:=HighRelative;
			TM_MovCmd_Speed:=30;
			TM_MovCmd_AccelTime:=200;
			TM_MovCmd_Blending:=100;
			TM_MovCmd_PrecisePos:=1;
			TM_MovCmd_RobotPose:='';
			TM_MovCmd_Command:='var_i=10';
			TM_MovCmd_ActivateExit:=TRUE;
			TM_MovCmd_CommandID:=2;
			TM_MovCmd_Execute:=FALSE;
			TM_MovCmd_ListenNode:='Listen1';
			IF (NOT TM_MovCmd_Done) AND (NOT TM_MovCmd_Error) THEN
				Stage:=182;
			END_IF;
		182:
			TM_MovCmd_Execute:=TRUE;
			IF TM_MovCmd_Done THEN
				Stage:=190;
			ELSIF TM_MovCmd_Error THEN
				Stage:=9999;
			END_IF;
		190:
			TM_MovCmd_Enable:=FALSE;
			MovementIndicatorStage:=Stage;
			IF (NOT TM_MovCmd_Done) AND (NOT TM_MovCmd_Error) AND (NOT TM_MovCmd_Busy) THEN
				Stage:=191;
			END_IF;	
		191:
			TM_MovCmd_Enable:=TRUE;
			TM_MovCmd_Movement:='Line';
			TM_MovCmd_DataFormat:='CPR';
			TM_MovCmd_Point:=PickPoint;
			TM_MovCmd_Speed:=30;
			TM_MovCmd_AccelTime:=200;
			TM_MovCmd_Blending:=100;
			TM_MovCmd_PrecisePos:=1;
			TM_MovCmd_RobotPose:='';
			TM_MovCmd_Command:='var_i=10';
			TM_MovCmd_ActivateExit:=FALSE;
			TM_MovCmd_CommandID:=1;
			TM_MovCmd_Execute:=FALSE;
			TM_MovCmd_ListenNode:='Listen1';
			IF (NOT TM_MovCmd_Done) AND (NOT TM_MovCmd_Error) THEN
				Stage:=192;
			END_IF;
		192:
			TM_MovCmd_Execute:=TRUE;
			IF TM_MovCmd_Done THEN
				Stage:=200;
			ELSIF TM_MovCmd_Error THEN
				Stage:=9999;
			END_IF;
		200:
			TM_MovCmd_Enable:=FALSE;
			IF (NOT TM_MovCmd_Done) AND (NOT TM_MovCmd_Error) AND (NOT TM_MovCmd_Busy) THEN
				Stage:=201;
			END_IF;	
		201:
			TM_MovCmd_Enable:=TRUE;
			TM_MovCmd_Movement:='Move_Line';
			TM_MovCmd_DataFormat:='CPP';
			TM_MovCmd_Point:=DownRelative;
			TM_MovCmd_Speed:=30;
			TM_MovCmd_AccelTime:=200;
			TM_MovCmd_Blending:=100;
			TM_MovCmd_PrecisePos:=1;
			TM_MovCmd_RobotPose:='';
			TM_MovCmd_Command:='var_i=10';
			TM_MovCmd_ActivateExit:=TRUE;
			TM_MovCmd_CommandID:=2;
			TM_MovCmd_Execute:=FALSE;
			TM_MovCmd_ListenNode:='Listen1';
			IF (NOT TM_MovCmd_Done) AND (NOT TM_MovCmd_Error) THEN
				Stage:=202;
			END_IF;
		202:
			TM_MovCmd_Execute:=TRUE;
			IF TM_MovCmd_Done THEN
				Stage:=210;
			ELSIF TM_MovCmd_Error THEN
				Stage:=9999;
			END_IF;
		210:
			TM_ChangeLoad_Enable:=FALSE;
			IF (NOT TM_ChangeLoad_Done) AND (NOT TM_ChangeLoad_Error) AND (NOT TM_ChangeLoad_Busy) THEN
				Stage:=211;
			END_IF;
		211:
			TM_ChangeLoad_Enable:=TRUE;	 
			TM_ChangeLoad_ActivateExit:=TRUE;
			TM_ChangeLoad_CommandID:=1;
			TM_ChangeLoad_Execute:=FALSE;
			TM_ChangeLoad_ListenNode:='Listen1';
			TM_ChangeLoad_Command:='var_i=20';
			TM_ChangeLoad_Payload:='0.2';
			IF (NOT TM_ChangeLoad_Done) AND (NOT TM_ChangeLoad_Error) THEN
				Stage:=212;
			END_IF;
		212:
			TM_ChangeLoad_Execute:=TRUE;
			IF TM_ChangeLoad_Done THEN
				Stage:=220;
			ELSIF TM_ChangeLoad_Error THEN
				Stage:=9999;
			END_IF;
		220:
			TM_MovCmd_Enable:=FALSE;
			IF (NOT TM_MovCmd_Done) AND (NOT TM_MovCmd_Error) AND (NOT TM_MovCmd_Busy) THEN
				Stage:=221;
			END_IF;
		221:
			TM_MovCmd_Enable:=TRUE;
			TM_MovCmd_Movement:='Move_Line';
			TM_MovCmd_DataFormat:='CPP';
			TM_MovCmd_Point:=HighRelative;
			TM_MovCmd_Speed:=30;
			TM_MovCmd_AccelTime:=200;
			TM_MovCmd_Blending:=100;
			TM_MovCmd_PrecisePos:=1;
			TM_MovCmd_RobotPose:='';
			TM_MovCmd_Command:='var_i=10';
			TM_MovCmd_ActivateExit:=TRUE;
			TM_MovCmd_CommandID:=2;
			TM_MovCmd_Execute:=FALSE;
			TM_MovCmd_ListenNode:='Listen1';
			IF (NOT TM_MovCmd_Done) AND (NOT TM_MovCmd_Error) THEN
				Stage:=222;
			END_IF;
		222:
			TM_MovCmd_Execute:=TRUE;
			IF TM_MovCmd_Done THEN
				Stage:=230;
			ELSIF TM_MovCmd_Error THEN
				Stage:=9999;
			END_IF;
		230:
			TM_MovCmd_Enable:=FALSE;
			MovementIndicatorStage:=Stage;
			IF (NOT TM_MovCmd_Done) AND (NOT TM_MovCmd_Error) AND (NOT TM_MovCmd_Busy) THEN
				Stage:=231;
			END_IF;
		231:
			TM_MovCmd_Enable:=TRUE;
			TM_MovCmd_Movement:='Line';
			TM_MovCmd_DataFormat:='CPR';
			TM_MovCmd_Point:=PalletThirdPoint;
			TM_MovCmd_Speed:=30;
			TM_MovCmd_AccelTime:=200;
			TM_MovCmd_Blending:=100;
			TM_MovCmd_PrecisePos:=1;
			TM_MovCmd_RobotPose:='';
			TM_MovCmd_Command:='var_i=10';
			TM_MovCmd_ActivateExit:=FALSE;
			TM_MovCmd_CommandID:=1;
			TM_MovCmd_Execute:=FALSE;
			TM_MovCmd_ListenNode:='Listen1';
			IF (NOT TM_MovCmd_Done) AND (NOT TM_MovCmd_Error) THEN
				Stage:=232;
			END_IF;
		232:
			TM_MovCmd_Execute:=TRUE;
			IF TM_MovCmd_Done THEN
				Stage:=240;
			ELSIF TM_MovCmd_Error THEN
				Stage:=9999;
			END_IF;
		240:
			TM_MovCmd_Enable:=FALSE;
			IF (NOT TM_MovCmd_Done) AND (NOT TM_MovCmd_Error) AND (NOT TM_MovCmd_Busy) THEN
				Stage:=241;
			END_IF;
		241:
			TM_MovCmd_Enable:=TRUE;
			TM_MovCmd_Movement:='Move_Line';
			TM_MovCmd_DataFormat:='CPP';
			TM_MovCmd_Point:=DownRelative;
			TM_MovCmd_Speed:=30;
			TM_MovCmd_AccelTime:=200;
			TM_MovCmd_Blending:=100;
			TM_MovCmd_PrecisePos:=1;
			TM_MovCmd_RobotPose:='';
			TM_MovCmd_Command:='var_i=10';
			TM_MovCmd_ActivateExit:=TRUE;
			TM_MovCmd_CommandID:=2;
			TM_MovCmd_Execute:=FALSE;
			TM_MovCmd_ListenNode:='Listen1';
			IF (NOT TM_MovCmd_Done) AND (NOT TM_MovCmd_Error) THEN
				Stage:=242;
			END_IF;
		242:
			TM_MovCmd_Execute:=TRUE;
			IF TM_MovCmd_Done THEN
				Stage:=250;
			ELSIF TM_MovCmd_Error THEN
				Stage:=9999;
			END_IF;
		250:
			TM_ChangeLoad_Enable:=FALSE;
			IF (NOT TM_ChangeLoad_Done) AND (NOT TM_ChangeLoad_Error) AND (NOT TM_ChangeLoad_Busy) THEN
				Stage:=251;
			END_IF;
		251:
			TM_ChangeLoad_Enable:=TRUE;	 
			TM_ChangeLoad_ActivateExit:=TRUE;
			TM_ChangeLoad_CommandID:=1;
			TM_ChangeLoad_Execute:=FALSE;
			TM_ChangeLoad_ListenNode:='Listen1';
			TM_ChangeLoad_Command:='var_i=30';
			TM_ChangeLoad_Payload:='0';
			IF (NOT TM_ChangeLoad_Done) AND (NOT TM_ChangeLoad_Error) THEN
				Stage:=252;
			END_IF;
		252:
			TM_ChangeLoad_Execute:=TRUE;
			IF TM_ChangeLoad_Done THEN
				Stage:=260;
			ELSIF TM_ChangeLoad_Error THEN
				Stage:=9999;
			END_IF;
		260:
			TM_MovCmd_Enable:=FALSE;
			IF (NOT TM_MovCmd_Done) AND (NOT TM_MovCmd_Error) AND (NOT TM_MovCmd_Busy) THEN
				Stage:=261;
			END_IF;
		261:
			TM_MovCmd_Enable:=TRUE;
			TM_MovCmd_Movement:='Move_Line';
			TM_MovCmd_DataFormat:='CPP';
			TM_MovCmd_Point:=HighRelative;
			TM_MovCmd_Speed:=30;
			TM_MovCmd_AccelTime:=200;
			TM_MovCmd_Blending:=100;
			TM_MovCmd_PrecisePos:=1;
			TM_MovCmd_RobotPose:='';
			TM_MovCmd_Command:='var_i=10';
			TM_MovCmd_ActivateExit:=TRUE;
			TM_MovCmd_CommandID:=2;
			TM_MovCmd_Execute:=FALSE;
			TM_MovCmd_ListenNode:='Listen1';
			IF (NOT TM_MovCmd_Done) AND (NOT TM_MovCmd_Error) THEN
				Stage:=262;
			END_IF;
		262:
			TM_MovCmd_Execute:=TRUE;
			IF TM_MovCmd_Done THEN
				Stage:=270;
			ELSIF TM_MovCmd_Error THEN
				Stage:=9999;
			END_IF;
		270:
			TM_MovCmd_Enable:=FALSE;
			MovementIndicatorStage:=Stage;
			IF (NOT TM_MovCmd_Done) AND (NOT TM_MovCmd_Error) AND (NOT TM_MovCmd_Busy) THEN
				Stage:=271;
			END_IF;
		271:
			TM_MovCmd_Enable:=TRUE;
			TM_MovCmd_Movement:='Line';
			TM_MovCmd_DataFormat:='CPR';
			TM_MovCmd_Point:=PickPoint;
			TM_MovCmd_Speed:=30;
			TM_MovCmd_AccelTime:=200;
			TM_MovCmd_Blending:=100;
			TM_MovCmd_PrecisePos:=1;
			TM_MovCmd_RobotPose:='';
			TM_MovCmd_Command:='var_i=10';
			TM_MovCmd_ActivateExit:=FALSE;
			TM_MovCmd_CommandID:=1;
			TM_MovCmd_Execute:=FALSE;
			TM_MovCmd_ListenNode:='Listen1';
			IF (NOT TM_MovCmd_Done) AND (NOT TM_MovCmd_Error) THEN
				Stage:=272;
			END_IF;
		272:
			TM_MovCmd_Execute:=TRUE;
			IF TM_MovCmd_Done THEN
				Stage:=280;
			ELSIF TM_MovCmd_Error THEN
				Stage:=9999;
			END_IF;
		280:
			TM_MovCmd_Enable:=FALSE;
			IF (NOT TM_MovCmd_Done) AND (NOT TM_MovCmd_Error) AND (NOT TM_MovCmd_Busy) THEN
				Stage:=281;
			END_IF;
		281:
			TM_MovCmd_Enable:=TRUE;
			TM_MovCmd_Movement:='Move_Line';
			TM_MovCmd_DataFormat:='CPP';
			TM_MovCmd_Point:=DownRelative;
			TM_MovCmd_Speed:=30;
			TM_MovCmd_AccelTime:=200;
			TM_MovCmd_Blending:=100;
			TM_MovCmd_PrecisePos:=1;
			TM_MovCmd_RobotPose:='';
			TM_MovCmd_Command:='var_i=10';
			TM_MovCmd_ActivateExit:=TRUE;
			TM_MovCmd_CommandID:=2;
			TM_MovCmd_Execute:=FALSE;
			TM_MovCmd_ListenNode:='Listen1';
			IF (NOT TM_MovCmd_Done) AND (NOT TM_MovCmd_Error) THEN
				Stage:=282;
			END_IF;
		282:
			TM_MovCmd_Execute:=TRUE;
			IF TM_MovCmd_Done THEN
				Stage:=290;
			ELSIF TM_MovCmd_Error THEN
				Stage:=9999;
			END_IF;
		290:
			TM_ChangeLoad_Enable:=FALSE;
			IF (NOT TM_ChangeLoad_Done) AND (NOT TM_ChangeLoad_Error) AND (NOT TM_ChangeLoad_Busy) THEN
				Stage:=291;
			END_IF;
		291:
			TM_ChangeLoad_Enable:=TRUE;	 
			TM_ChangeLoad_ActivateExit:=TRUE;
			TM_ChangeLoad_CommandID:=1;
			TM_ChangeLoad_Execute:=FALSE;
			TM_ChangeLoad_ListenNode:='Listen1';
			TM_ChangeLoad_Command:='var_i=20';
			TM_ChangeLoad_Payload:='0.2';
			IF (NOT TM_ChangeLoad_Done) AND (NOT TM_ChangeLoad_Error) THEN
				Stage:=292;
			END_IF;
		292:
			TM_ChangeLoad_Execute:=TRUE;
			IF TM_ChangeLoad_Done THEN
				Stage:=300;
			ELSIF TM_ChangeLoad_Error THEN
				Stage:=9999;
			END_IF;
		300:
			TM_MovCmd_Enable:=FALSE;
			IF (NOT TM_MovCmd_Done) AND (NOT TM_MovCmd_Error) AND (NOT TM_MovCmd_Busy) THEN
				Stage:=301;
			END_IF;
		301:
			TM_MovCmd_Enable:=TRUE;
			TM_MovCmd_Movement:='Move_Line';
			TM_MovCmd_DataFormat:='CPP';
			TM_MovCmd_Point:=HighRelative;
			TM_MovCmd_Speed:=30;
			TM_MovCmd_AccelTime:=200;
			TM_MovCmd_Blending:=100;
			TM_MovCmd_PrecisePos:=1;
			TM_MovCmd_RobotPose:='';
			TM_MovCmd_Command:='var_i=10';
			TM_MovCmd_ActivateExit:=TRUE;
			TM_MovCmd_CommandID:=2;
			TM_MovCmd_Execute:=FALSE;
			TM_MovCmd_ListenNode:='Listen1';
			IF (NOT TM_MovCmd_Done) AND (NOT TM_MovCmd_Error) THEN
				Stage:=302;
			END_IF;
		302:
			TM_MovCmd_Execute:=TRUE;
			IF TM_MovCmd_Done THEN
				Stage:=310;
			ELSIF TM_MovCmd_Error THEN
				Stage:=9999;
			END_IF;
		310:
			TM_MovCmd_Enable:=FALSE;
			MovementIndicatorStage:=Stage;
			IF (NOT TM_MovCmd_Done) AND (NOT TM_MovCmd_Error) AND (NOT TM_MovCmd_Busy) THEN
				Stage:=311;
			END_IF;
		311:
			TM_MovCmd_Enable:=TRUE;
			TM_MovCmd_Movement:='Line';
			TM_MovCmd_DataFormat:='CPR';
			TM_MovCmd_Point:=PalletFourthPoint;
			TM_MovCmd_Speed:=30;
			TM_MovCmd_AccelTime:=200;
			TM_MovCmd_Blending:=100;
			TM_MovCmd_PrecisePos:=1;
			TM_MovCmd_RobotPose:='';
			TM_MovCmd_Command:='var_i=10';
			TM_MovCmd_ActivateExit:=FALSE;
			TM_MovCmd_CommandID:=1;
			TM_MovCmd_Execute:=FALSE;
			TM_MovCmd_ListenNode:='Listen1';
			IF (NOT TM_MovCmd_Done) AND (NOT TM_MovCmd_Error) THEN
				Stage:=312;
			END_IF;
		312:
			TM_MovCmd_Execute:=TRUE;
			IF TM_MovCmd_Done THEN
				Stage:=320;
			ELSIF TM_MovCmd_Error THEN
				Stage:=9999;
			END_IF;
		320:
			TM_MovCmd_Enable:=FALSE;
			IF (NOT TM_MovCmd_Done) AND (NOT TM_MovCmd_Error) AND (NOT TM_MovCmd_Busy) THEN
				Stage:=321;
			END_IF;
		321:
			TM_MovCmd_Enable:=TRUE;
			TM_MovCmd_Movement:='Move_Line';
			TM_MovCmd_DataFormat:='CPP';
			TM_MovCmd_Point:=DownRelative;
			TM_MovCmd_Speed:=30;
			TM_MovCmd_AccelTime:=200;
			TM_MovCmd_Blending:=100;
			TM_MovCmd_PrecisePos:=1;
			TM_MovCmd_RobotPose:='';
			TM_MovCmd_Command:='var_i=10';
			TM_MovCmd_ActivateExit:=TRUE;
			TM_MovCmd_CommandID:=2;
			TM_MovCmd_Execute:=FALSE;
			TM_MovCmd_ListenNode:='Listen1';
			IF (NOT TM_MovCmd_Done) AND (NOT TM_MovCmd_Error) THEN
				Stage:=322;
			END_IF;
		322:
			TM_MovCmd_Execute:=TRUE;
			IF TM_MovCmd_Done THEN
				Stage:=330;
			ELSIF TM_MovCmd_Error THEN
				Stage:=9999;
			END_IF;
		330:
			TM_ChangeLoad_Enable:=FALSE;
			IF (NOT TM_ChangeLoad_Done) AND (NOT TM_ChangeLoad_Error) AND (NOT TM_ChangeLoad_Busy) THEN
				Stage:=331;
			END_IF;
		331:
			TM_ChangeLoad_Enable:=TRUE;	 
			TM_ChangeLoad_ActivateExit:=TRUE;
			TM_ChangeLoad_CommandID:=1;
			TM_ChangeLoad_Execute:=FALSE;
			TM_ChangeLoad_ListenNode:='Listen1';
			TM_ChangeLoad_Command:='var_i=30';
			TM_ChangeLoad_Payload:='0';
			IF (NOT TM_ChangeLoad_Done) AND (NOT TM_ChangeLoad_Error) THEN
				Stage:=332;
			END_IF;
		332:
			TM_ChangeLoad_Execute:=TRUE;
			IF TM_ChangeLoad_Done THEN
				Stage:=340;
			ELSIF TM_ChangeLoad_Error THEN
				Stage:=9999;
			END_IF;
		340:
			TM_MovCmd_Enable:=FALSE;
			IF (NOT TM_MovCmd_Done) AND (NOT TM_MovCmd_Error) AND (NOT TM_MovCmd_Busy) THEN
				Stage:=341;
			END_IF;
		341:
			TM_MovCmd_Enable:=TRUE;
			TM_MovCmd_Movement:='Move_Line';
			TM_MovCmd_DataFormat:='CPP';
			TM_MovCmd_Point:=HighRelative;
			TM_MovCmd_Speed:=30;
			TM_MovCmd_AccelTime:=200;
			TM_MovCmd_Blending:=100;
			TM_MovCmd_PrecisePos:=1;
			TM_MovCmd_RobotPose:='';
			TM_MovCmd_Command:='var_i=10';
			TM_MovCmd_ActivateExit:=TRUE;
			TM_MovCmd_CommandID:=2;
			TM_MovCmd_Execute:=FALSE;
			TM_MovCmd_ListenNode:='Listen1';
			IF (NOT TM_MovCmd_Done) AND (NOT TM_MovCmd_Error) THEN
				Stage:=342;
			END_IF;
		342:
			TM_MovCmd_Execute:=TRUE;
			IF TM_MovCmd_Done THEN
				Stage:=350;
			ELSIF TM_MovCmd_Error THEN
				Stage:=9999;
			END_IF;
		350:
			TM_MovCmd_Enable:=FALSE;
			MovementIndicatorStage:=Stage;
			IF (NOT TM_MovCmd_Done) AND (NOT TM_MovCmd_Error) AND (NOT TM_MovCmd_Busy) THEN
				Stage:=351;
			END_IF;
		351:		
			TM_MovCmd_Enable:=TRUE;
			TM_MovCmd_Movement:='Line';
			TM_MovCmd_DataFormat:='CPR';
			TM_MovCmd_Point:=StartPoint;
			TM_MovCmd_Speed:=30;
			TM_MovCmd_AccelTime:=200;
			TM_MovCmd_Blending:=100;
			TM_MovCmd_PrecisePos:=1;
			TM_MovCmd_RobotPose:='';
			TM_MovCmd_Command:='var_i=10';
			TM_MovCmd_ActivateExit:=TRUE;
			TM_MovCmd_CommandID:=1;
			TM_MovCmd_Execute:=FALSE;
			TM_MovCmd_ListenNode:='Listen1';
			IF (NOT TM_MovCmd_Done) AND (NOT TM_MovCmd_Error) THEN
				Stage:=352;
			END_IF;
		352:
			TM_MovCmd_Execute:=TRUE;
			IF TM_MovCmd_Done THEN
				Stage:=0;
			ELSIF TM_MovCmd_Error THEN
				Stage:=9999;
			END_IF;
				
	END_CASE;
	
END_IF;

TM_MovCmd_Instance(
	Done=>TM_MovCmd_Done,
	Busy=>TM_MovCmd_Busy,
	Error=>TM_MovCmd_Error,
	ErrorID=>TM_MovCmd_ErrorID,
	Execute:=TM_MovCmd_Execute,
	RobotID:=ListenNode_Connect_TCP_Socket,
	Movement:=TM_MovCmd_Movement,
	DataFormat:=TM_MovCmd_DataFormat,
	Point:=TM_MovCmd_Point,
	Speed:=TM_MovCmd_Speed,
	AccelTime:=TM_MovCmd_AccelTime,
	Blending:=TM_MovCmd_Blending,
	PrecisePos:=TM_MovCmd_PrecisePos,
	RobotPose:=TM_MovCmd_RobotPose,
	Command:=TM_MovCmd_Command,  
	ActivateExit:=TM_MovCmd_ActivateExit,
	CommandID:=TM_MovCmd_CommandID,
	TimeOut:=T#3600s,
	ListenNode:=TM_MovCmd_ListenNode,
	TimeOutET=>TM_MovCmd_TimeOutET,
	Enable:=TM_MovCmd_Enable
);

TM_ChangeTCP_Instance(
	Enable:=TM_ChangeTCP_Enable,
	Execute:=TM_ChangeTCP_Execute,
	RobotID:=ListenNode_Connect_TCP_Socket,
	TCP:=TM_ChangeTCP_TCP,
	Weight:=TM_ChangeTCP_Weight,
	MomInertia:=TM_ChangeTCP_MomInertia,
	RefFrame:=TM_ChangeTCP_RefFrame,
	Command:=TM_ChangeTCP_Command,
	ActivateExit:=TM_ChangeTCP_ActivateExit,
	ListenNode:=TM_ChangeTCP_ListenNode,
	TimeOut:=T#3600s,
	CommandID:=TM_ChangeTCP_CommandID,
	Done=>TM_ChangeTCP_Done,
	Busy=>TM_ChangeTCP_Busy,
	Error=>TM_ChangeTCP_Error,
	ErrorID=>TM_ChangeTCP_ErrorID,
	TimeOutET=>TM_ChangeTCP_TimeOutET
);

TM_ChangeLoad_Instance(
	Enable:=TM_ChangeLoad_Enable,
	Execute:=TM_ChangeLoad_Execute,
	RobotID:=ListenNode_Connect_TCP_Socket,
	Payload:=TM_ChangeLoad_Payload,
	Command:=TM_ChangeLoad_Command,
	ActivateExit:=TM_ChangeLoad_ActivateExit,
	ListenNode:=TM_ChangeLoad_ListenNode,
	TimeOut:=T#3600s,
	CommandID:=TM_ChangeLoad_CommandID,
	Done=>TM_ChangeLoad_Done,
	Busy=>TM_ChangeLoad_Busy,
	Error=>TM_ChangeLoad_Error,
	ErrorID=>TM_ChangeLoad_ErrorID,
	TimeOutET=>TM_ChangeLoad_TimeOutET
);

TM_CircleCmd_Instance(
	Enable:=TM_CircleCmd_Enable,
	Execute:=TM_CircleCmd_Execute,
	RobotID:=ListenNode_Connect_TCP_Socket,
	DataFormat:=TM_CircleCmd_DataFormat,
	ArcPoint:=TM_CircleCmd_ArcPoint,
	EndArcPoint:=TM_CircleCmd_EndArcPoint,
	Speed:=TM_CircleCmd_Speed,
	AccelTime:=TM_CircleCmd_AccelTime,
	Blending:=TM_CircleCmd_Blending,
	ArcAngle:=TM_CircleCmd_ArcAngle,
	PrecisePos:=TM_CircleCmd_PrecisePos,
	Command:=TM_CircleCmd_Command,
	ActivateExit:=TM_CircleCmd_ActivateExit,
	ListenNode:=TM_CircleCmd_ListenNode,
	TimeOut:=T#3600s,
	CommandID:=TM_CircleCmd_CommandID,
	Done=>TM_CircleCmd_Done,
	Busy=>TM_CircleCmd_Busy,
	Error=>TM_CircleCmd_Error,
	ErrorID=>TM_CircleCmd_ErrorID,
	TimeOutET=>TM_CircleCmd_TimeOutET
);

TM_ChangeBase_Instance(
	Enable:=TM_ChangeBase_Enable,
	Execute:=TM_ChangeBase_Execute,
	RobotID:=ListenNode_Connect_TCP_Socket,
	Base:=TM_ChangeBase_Base,
	Command:=TM_ChangeBase_Command,
	ActivateExit:=TM_ChangeBase_ActivateExit,
	ListenNode:=TM_ChangeBase_ListenNode,
	TimeOut:=T#3600s,
	CommandID:=TM_ChangeBase_CommandID,
	Done=>TM_ChangeBase_Done,
	Busy=>TM_ChangeBase_Busy,
	Error=>TM_ChangeBase_Error,
	ErrorID=>TM_ChangeBase_ErrorID,
	TimeOutET=>TM_ChangeBase_TimeOutET
);
END_PROGRAM